# EPICS substitutions: epics_iocs/GaussMeter/group5App/Db/user.substitutions
# Example substitutions file

file "db/circle.db" {
    { user = "epics" }
}

file "db/dbExample1.db" {
    { user = "epics" }
}

file db/dbExample2.db {
    pattern { user, no, scan }
        { "epics", 1, "1 second" }
        { "epics", 2, "2 second" }
        { "epics", 3, "5 second" }
}
